// Mitsubishi GX Works2 project: FX1N_Modbus_RTU_V02   PLC: FX1N/FX1NC

PROGRAM MAIN
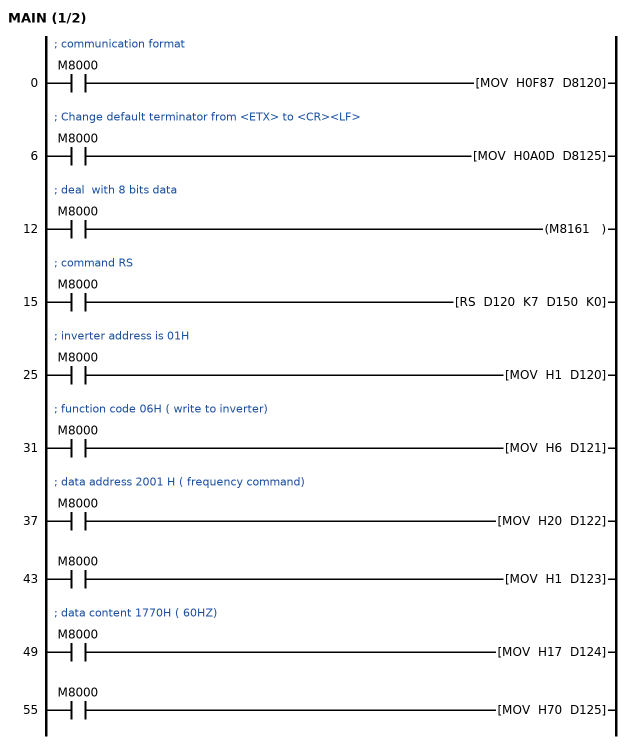
; communication format
0     LD      M8000
      MOV     H0F87 D8120
; Change default terminator from <ETX> to <CR><LF>
6     LD      M8000
      MOV     H0A0D D8125
; deal  with 8 bits data
12    LD      M8000
      OUT     M8161
; command RS
15    LD      M8000
      RS      D120 K7 D150 K0
; inverter address is 01H
25    LD      M8000
      MOV     H1 D120
; function code 06H ( write to inverter)
31    LD      M8000
      MOV     H6 D121
; data address 2001 H ( frequency command)
37    LD      M8000
      MOV     H20 D122
43    LD      M8000
      MOV     H1 D123
; data content 1770H ( 60HZ)
49    LD      M8000
      MOV     H17 D124
55    LD      M8000
      MOV     H70 D125
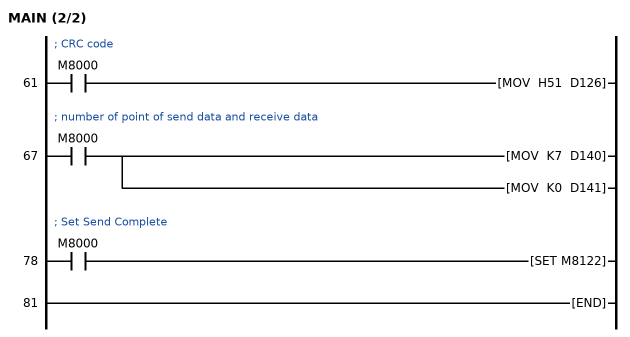
; CRC code
61    LD      M8000
      MOV     H51 D126
; number of point of send data and receive data
67    LD      M8000
      MOV     K7 D140
      MOV     K0 D141
; Set Send Complete
78    LD      M8000
      SET     M8122
81    END
END_PROGRAM
